// TwinCAT 3 PLC project TCP_IP
// ProgramVersion: 3.1.4023.0
// libraries:
//   Tc2_Standard, * (Beckhoff Automation GmbH)
//   Tc2_System, * (Beckhoff Automation GmbH)
//   Tc2_TcpIp, * (Beckhoff Automation GmbH)
//   Tc2_Utilities, * (Beckhoff Automation GmbH)
//   Tc3_JsonXml, * (Beckhoff Automation GmbH)
//   Tc3_Module, * (Beckhoff Automation GmbH)
// project tree:
//   / PlcTask.TcTTO (not stored)
//   POUs/ MAIN.TcPOU, tcp_ip.TcPOU

// ---- POUs/MAIN.TcPOU
PROGRAM MAIN
VAR
END_VAR

tcp_ip();

END_PROGRAM

// ---- POUs/tcp_ip.TcPOU
PROGRAM tcp_ip
VAR
	bConnect : BOOL;
	bRecieve : BOOL;
	FB_create : FB_SocketUdpCreate;
	FB_Recieve: FB_SocketUdpReceiveFrom;
	FB_close  : FB_SocketClose;
	data: ARRAY[0..5000] OF BYTE;
END_VAR

FB_create(
	sSrvNetId:= , 							//Lokaal netwerk (mag leeg blijven)
	sLocalHost:= '192.168.1.158', 			//Eigen ip van de PC en ingesteld in de gateway
	nLocalPort:= 25565,						//Ingesteld op de gateway
	bExecute:= bConnect,					//Trigger voor functieblok
	tTimeout:= T#10S);


FB_Recieve(
	sSrvNetId:= , 									//Lokaal netwerk (mag leeg blijven)
	hSocket:= FB_create.hSocket,					 
	cbLen:= SIZEOF(data), 							//Kijkt naar de lengte van het bericht
	pDest:= ADR(data), 								//Plaat waar de het bericht wordt opgeslaan
	bExecute:= NOT FB_recieve.bBusy AND bRecieve, 	//Trigger voor functieblok
	tTimeout:= T#10S);
	
FB_close(
	sSrvNetId:= , 							//Lokaal netwerk (mag leeg blijven)
	hSocket:= FB_create.hSocket, 			
	bExecute:= NOT bConnect, 				//Sluiten van de connectie 
	tTimeout:= T#1S);

END_PROGRAM
